FUNCTION_BLOCK EmergencyManagement_HMI (* Service Interface Function Block Type *)
  (* Standard: 61499-2 *)
  (* Version 0.0, 7/4/2026, Schneider Electric, template *)
  PACKAGE SE.Nereda;
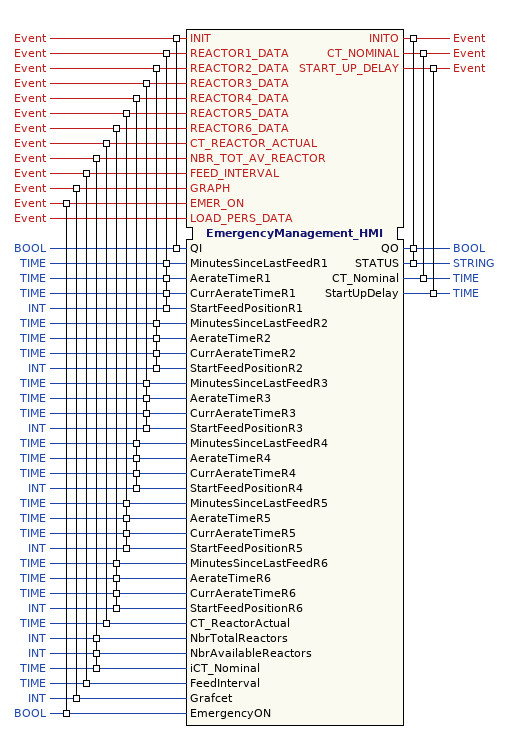
  EVENT_INPUT
    INIT WITH QI;
    REACTOR1_DATA WITH MinutesSinceLastFeedR1, AerateTimeR1, StartFeedPositionR1, CurrAerateTimeR1;
    REACTOR2_DATA WITH MinutesSinceLastFeedR2, AerateTimeR2, StartFeedPositionR2, CurrAerateTimeR2;
    REACTOR3_DATA WITH MinutesSinceLastFeedR3, AerateTimeR3, StartFeedPositionR3, CurrAerateTimeR3;
    REACTOR4_DATA WITH MinutesSinceLastFeedR4, AerateTimeR4, StartFeedPositionR4, CurrAerateTimeR4;
    REACTOR5_DATA WITH MinutesSinceLastFeedR5, AerateTimeR5, StartFeedPositionR5, CurrAerateTimeR5;
    REACTOR6_DATA WITH MinutesSinceLastFeedR6, AerateTimeR6, StartFeedPositionR6, CurrAerateTimeR6;
    CT_REACTOR_ACTUAL WITH CT_ReactorActual;
    NBR_TOT_AV_REACTOR WITH NbrTotalReactors, NbrAvailableReactors, iCT_Nominal;
    FEED_INTERVAL WITH FeedInterval;
    GRAPH WITH Grafcet;
    EMER_ON WITH EmergencyON;
    LOAD_PERS_DATA;
  END_EVENT
  EVENT_OUTPUT
    INITO WITH QO, STATUS;
    CT_NOMINAL WITH CT_Nominal;
    START_UP_DELAY WITH StartUpDelay;
  END_EVENT
  VAR_INPUT
    QI : BOOL;
    MinutesSinceLastFeedR1 : TIME;
    AerateTimeR1 : TIME;
    CurrAerateTimeR1 : TIME;
    StartFeedPositionR1 : INT;
    MinutesSinceLastFeedR2 : TIME;
    AerateTimeR2 : TIME;
    CurrAerateTimeR2 : TIME;
    StartFeedPositionR2 : INT;
    MinutesSinceLastFeedR3 : TIME;
    AerateTimeR3 : TIME;
    CurrAerateTimeR3 : TIME;
    StartFeedPositionR3 : INT;
    MinutesSinceLastFeedR4 : TIME;
    AerateTimeR4 : TIME;
    CurrAerateTimeR4 : TIME;
    StartFeedPositionR4 : INT;
    MinutesSinceLastFeedR5 : TIME;
    AerateTimeR5 : TIME;
    CurrAerateTimeR5 : TIME;
    StartFeedPositionR5 : INT;
    MinutesSinceLastFeedR6 : TIME;
    AerateTimeR6 : TIME;
    CurrAerateTimeR6 : TIME;
    StartFeedPositionR6 : INT;
    CT_ReactorActual : TIME;
    NbrTotalReactors : INT;
    NbrAvailableReactors : INT;
    iCT_Nominal : TIME;
    FeedInterval : TIME;
    Grafcet : INT;
    EmergencyON : BOOL;
  END_VAR
  VAR_OUTPUT
    QO : BOOL; (* Event Output Qualifier *)
    STATUS : STRING; (* Service Status *)
    CT_Nominal : TIME; (* Nominal cycle time *)
    StartUpDelay : TIME;
  END_VAR
  SERVICE /
    SEQUENCE 
    END_SEQUENCE
  END_SERVICE
END_FUNCTION_BLOCK
